// TwinCAT 3 PLC project Plc
// ProgramVersion: 3.1.4024.0
// libraries:
//   Tc2_Standard, * (Beckhoff Automation GmbH)
//   Tc2_System, * (Beckhoff Automation GmbH)
//   Tc3_Module, * (Beckhoff Automation GmbH)
// project tree:
//   / PlcTask.TcTTO, PlcTask2.TcTTO
//   POUs/ MAIN.TcPOU, MAIN_2.TcPOU
// real-time tasks:
//   TASK PlcTask: cycle T#10ms, priority 20, ADS port 350
//   TASK PlcTask2: cycle T#5ms, priority 1, ADS port 351
// I/O:
//   DEVICE Dispositivo 1 (EtherCAT), AmsNetId 192.168.19.131.2.1
//     Terminale 1 (EK1200) [EK1200-5000 EtherCAT Power supply (2A E-Bus)]

CONFIGURATION Plc
    RESOURCE PLC ON TwinCAT3
        TASK PlcTask(INTERVAL := T#10ms, PRIORITY := 20);
        TASK PlcTask2(INTERVAL := T#5ms, PRIORITY := 1);
        PROGRAM MAIN WITH PlcTask : MAIN;
        PROGRAM MAIN_2 WITH PlcTask2 : MAIN_2;
    END_RESOURCE
END_CONFIGURATION

// ---- POUs/MAIN.TcPOU
PROGRAM MAIN
VAR
	test	: DINT;
END_VAR

test:=test+1;

END_PROGRAM

// ---- POUs/MAIN_2.TcPOU
PROGRAM MAIN_2
VAR
	test2	: DINT;
END_VAR

test2:=test2+1;

END_PROGRAM
